(* PLC project Tc3_EventLogger.GetJsonAttribute Demo, tc3-libraries-kb TwinCAT 3.1 *)
(* stored: creationDateTime 2026-05-11T01:00:00, modificationDateTime 2026-05-11T01:00:00 *)

PROGRAM P_Demo_GetJsonAttribute
  VAR
    fbAlarm : FB_TcAlarm;  (* alarm 实例 *)
    sJsonAttribute : STRING;  (* JSON 输出缓冲 *)
    bRead : BOOL := FALSE;  (* 上升沿触发读取 *)
    bReadPrev : BOOL;  (* 边沿检测 *)
    hr : HRESULT;  (* 返回值监视 *)
  END_VAR

// =============================================================================
// 场景：读取 alarm 的 JSON 属性以提取 batch id
// 价值：一句调用拿到 JSON 字符串供后续解析
// 验证：先用 SetJsonAttribute 写一个 JSON，再用本方法读取，sJsonAttribute 应等于写入值
// 验证步骤：
//   1. 右键 PLC 项目 → Import PLCopenXML → 选本文件
//   2. 引用 Tc3_EventLogger（System → References → Add library）
//   3. 编译 → 登录 → 运行；按 verify 注释里给出的在线写值操作
// =============================================================================

IF bRead AND NOT bReadPrev THEN
    hr := fbAlarm.GetJsonAttribute(sJsonAttribute := sJsonAttribute);
END_IF;
bReadPrev := bRead;
END_PROGRAM
